FUNCTION_BLOCK L2_Simple_SFC EXTENDS L1_ControllerBase_SFC
// Grafcet simple para los detectores fotoeléctrico e inductivo

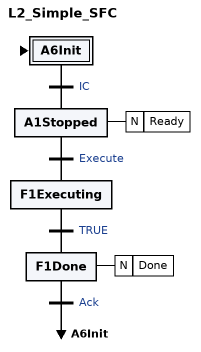
INITIAL_STEP A6Init:
END_STEP
TRANSITION FROM A6Init TO A1Stopped
    := IC;
END_TRANSITION
STEP A1Stopped:
    Ready(N);
END_STEP
TRANSITION FROM A1Stopped TO F1Executing
    := Execute;
END_TRANSITION
STEP F1Executing:
END_STEP
TRANSITION FROM F1Executing TO F1Done
    := TRUE;
END_TRANSITION
STEP F1Done:
    Done(N);
END_STEP
TRANSITION FROM F1Done TO A6Init
    := Ack;
END_TRANSITION

END_FUNCTION_BLOCK

(* stored: Version 1.1.0.1, ProductVersion 3.1.4024.11
   POU L2_Simple_SFC: Id {88f7459f-e3cd-4931-a3a9-314c818d385e}, SpecialFunc None *)
